PROGRAM Control_FBD
VAR
	
	ixPulse			AT %I*:	BOOL; 		(* PULS button *)
	ixStart			AT %I*:	BOOL; 		(* START switch *)
	ixSetLevel		AT %I*:	BOOL; 		(* NIVÅ switch *)
	ixLevel3		AT %I*:	BOOL; 		(* Sensor for level 3 *)
	ixLevel2		AT %I*:	BOOL; 		(* Sensor for level 2 *)
	ixLevel1		AT %I*:	BOOL; 		(* Sensor for level 1 *)
	ixNotEmpty		AT %I*:	BOOL; 		(* Sensor for not empty *)
	ixTempOk		AT %I*:	BOOL; 		(* Temp sensor *)

	qxForw			AT %Q*:	BOOL; 		(* Washer cylinder forward *)
	qxBack			AT %Q*:	BOOL; 		(* Washer cylinder back *)
	qxSpin			AT %Q*:	BOOL; 		(* Washer cylinder spin *)
	qxFill			AT %Q*:	BOOL; 		(* Fill water *)
	qxDrain			AT %Q*:	BOOL; 		(* Drain water *)
	qxHeat			AT %Q*:	BOOL; 		(* Heat water *)
	qxDispBit1		AT %Q*:	BOOL; 		(* Display bit 1 *)
	qxDispBit2		AT %Q*:	BOOL; 		(* Display bit 2 *)
	CTU_0: CTU;

	time_to_drain: BOOL;
	maxFill: CTU;
END_VAR

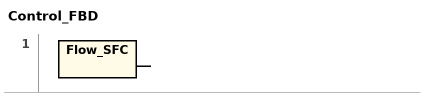
// NETWORK 1
Flow_SFC();

ACTION Flow_SFC:
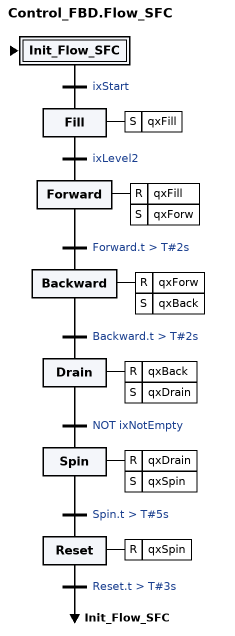
INITIAL_STEP Init_Flow_SFC:
END_STEP
TRANSITION FROM Init_Flow_SFC TO Fill
    := ixStart;
END_TRANSITION
STEP Fill:
    qxFill(S);
END_STEP
TRANSITION FROM Fill TO Forward
    := ixLevel2;
END_TRANSITION
STEP Forward:
    qxFill(R);
    qxForw(S);
END_STEP
TRANSITION FROM Forward TO Backward
    := Forward.t > T#2s;
END_TRANSITION
STEP Backward:
    qxForw(R);
    qxBack(S);
END_STEP
TRANSITION FROM Backward TO Drain
    := Backward.t > T#2s;
END_TRANSITION
STEP Drain:
    qxBack(R);
    qxDrain(S);
END_STEP
TRANSITION FROM Drain TO Spin
    := NOT ixNotEmpty;
END_TRANSITION
STEP Spin:
    qxDrain(R);
    qxSpin(S);
END_STEP
TRANSITION FROM Spin TO Reset
    := Spin.t > T#5s;
END_TRANSITION
STEP Reset:
    qxSpin(R);
END_STEP
TRANSITION FROM Reset TO Init_Flow_SFC
    := Reset.t > T#3s;
END_TRANSITION
END_ACTION

ACTION maxFilling:
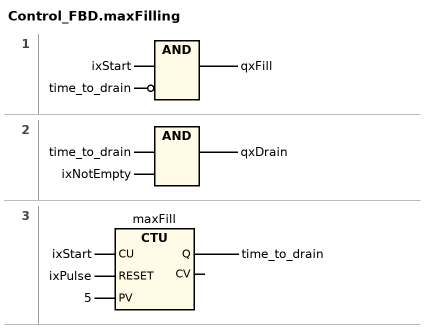
// NETWORK 1
qxFill := ixStart AND NOT time_to_drain;

// NETWORK 2
qxDrain := time_to_drain AND ixNotEmpty;

// NETWORK 3
maxFill(CU := ixStart, RESET := ixPulse, PV := 5); // CTU
time_to_drain := maxFill.Q;
END_ACTION

END_PROGRAM

(* stored: Version 1.1.0.1, ProductVersion 3.1.4024.12
   POU Control_FBD: Id {84d3f40d-a0f6-423e-bc58-eeabb716185d}, SpecialFunc None
   Action Flow_SFC: Id {ae57ce22-386b-4db0-a9c6-c4881053702a}
   Action maxFilling: Id {cd4d31ad-dc60-4aa2-aacf-d01c9f49ffb6} *)
